// TIA Portal V19 export
TYPE "LEXCHANGETRAY_typeTraySpecification"
// stored: Access Published
   STRUCT
      traySize : Int;   // 24,36
      rowCellsSpacing : LReal;   // 行与行之间电芯间距
      rows : Int := 2;   // 行数
      trayType : Int;   // 0:constraint 1:plastic
   END_STRUCT;
END_TYPE
